// TIA Portal V17 export
// export: Created 2022-03-16T18:47:26.5380485Z, ExportSetting WithDefaults, DisplayName Totally Integrated Automation Portal, DisplayVersion V17, DisplayName TIA Portal Openness, DisplayVersion V17, DisplayName TIA Portal Version Control Interface, DisplayVersion V17, DisplayName STEP 7 Professional, DisplayVersion V17, DisplayName STEP 7 Safety, DisplayVersion V17, DisplayName WinCC Advanced / Unified PC, DisplayVersion V17
FUNCTION_BLOCK "EM00_CM05_Conveyor"   // FB2, LAD
TITLE = EM00_CM04 / EM00_CM05
{ S7_Optimized_Access := 'TRUE' }
AUTHOR : tech.team.motioncontrol@siemens.com
FAMILY : CPG
VERSION : 1.1
// Support: tech.team.motioncontrol@siemens.com
// stored: AutoNumber true, IsIECCheckEnabled false, IsRetainMemResEnabled false, MemoryReserve 100, SetENOAutomatically false, UDAEnableTagReadback false
   VAR
      statDummyBool { ExternalAccessible := 'False'; ExternalVisible := 'False'; ExternalWritable := 'False'} : Bool;   // dummy bool - placeholder
   END_VAR
BEGIN

REGION Network 1: *** Begin the Setpoint Management Information Section ***
END_REGION

REGION Network 2: *** Begin the Logic Section ***
END_REGION

REGION Network 3: *** Begin the Event Information Section ***
END_REGION

REGION Network 4: *** Begin the State Model Status Feedback Section ***
END_REGION

REGION Network 5: *** Call the PackML Module Initialize Logic ***
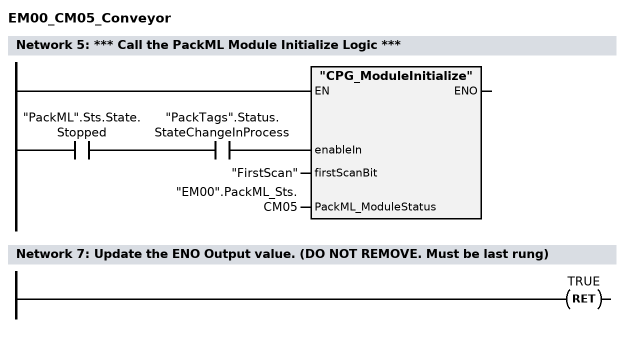
   RUNG wire#powerrail
      "CPG_ModuleInitialize"(enableIn := wire#w1, firstScanBit := "FirstScan", PackML_ModuleStatus := "EM00".PackML_Sts.CM05)
   END_RUNG
   RUNG wire#powerrail
      Contact( "PackML".Sts.State.Stopped )
      Contact( "PackTags".Status.StateChangeInProcess )
   END_RUNG wire#w1
   // the same network as SCL:
   "CPG_ModuleInitialize"(enableIn := "PackML".Sts.State.Stopped AND "PackTags".Status.StateChangeInProcess,
                          firstScanBit := "FirstScan",
                          PackML_ModuleStatus := "EM00".PackML_Sts.CM05);
END_REGION

REGION Network 7: Update the ENO Output value. (DO NOT REMOVE. Must be last rung)
   RUNG wire#powerrail
      ReturnCoil( TRUE )
   END_RUNG
   // the same network as SCL:
   ENO := TRUE;
   RETURN;
END_REGION
END_FUNCTION_BLOCK
